FUNCTION TryConvert_BOOL_TO_STRING : BOOL
VAR_INPUT
	in : BOOL;
	out : REFERENCE TO STRING;
END_VAR

out := BOOL_TO_STRING(in);
TryConvert_BOOL_TO_STRING := TRUE;

END_FUNCTION

(* stored: Version 1.1.0.1, ProductVersion 3.1.4024.12
   POU TryConvert_BOOL_TO_STRING: Id {8096e369-4428-4d4c-b536-ff4218bfa109}, SpecialFunc None *)
